(* IEC 61131-3 sources: Elmo_Master/Lasal_PRG/Elmo_EtherCAT_Test_4Axis/Class/Byte_to_Bit, 1 file *)

(* ---- Byte_to_Bit.st ---- *)
(*!
<Class
	Name               = "Byte_to_Bit"
	Revision           = "0.0"
	RealtimeTask       = "false"
	CyclicTask         = "false"
	DefCyclictime      = "1 ms"
	BackgroundTask     = "false"
	Sigmatek           = "false"
	OSInterface        = "false"
	HighPriority       = "false"
	Automatic          = "false"
	UpdateMode         = "Prescan"
	SharedCommandTable = "true"
	Objectsize         = "(300,120)">
	<Channels>
		<Server Name="bit1" Visualized="false" Initialize="false" WriteProtected="true" Retentive="false"/>
		<Server Name="bit2" Visualized="false" Initialize="false" WriteProtected="true" Retentive="false"/>
		<Server Name="bit3" Visualized="false" Initialize="false" WriteProtected="true" Retentive="false"/>
		<Server Name="bit4" Visualized="false" Initialize="false" WriteProtected="true" Retentive="false"/>
		<Server Name="bit5" Visualized="false" Initialize="false" WriteProtected="true" Retentive="false"/>
		<Server Name="bit6" Visualized="false" Initialize="false" WriteProtected="true" Retentive="false"/>
		<Server Name="bit7" Visualized="false" Initialize="false" WriteProtected="true" Retentive="false"/>
		<Server Name="bit8" Visualized="false" Initialize="false" WriteProtected="true" Retentive="false"/>
		<Server Name="ClassSvr" Visualized="false" Initialize="false" WriteProtected="true" Retentive="false"/>
		<Client Name="fromByte" Required="true" Internal="false"/>
	</Channels>
</Class>
*)
Byte_to_Bit : CLASS
  //Servers:
	ClassSvr 	: SvrChCmd_DINT;
	bit1 	: SvrCh_DINT;
	bit2 	: SvrCh_DINT;
	bit3 	: SvrCh_DINT;
	bit4 	: SvrCh_DINT;
	bit5 	: SvrCh_DINT;
	bit6 	: SvrCh_DINT;
	bit7 	: SvrCh_DINT;
	bit8 	: SvrCh_DINT;
  //Clients:
	fromByte 	: CltCh_BDINT;
  //Variables:
  //Functions:

	FUNCTION ReadByte;

	FUNCTION VIRTUAL GLOBAL bit1::Read
		VAR_OUTPUT
			output (EAX) 	: DINT;
		END_VAR;

	FUNCTION VIRTUAL GLOBAL bit2::Read
		VAR_OUTPUT
			output (EAX) 	: DINT;
		END_VAR;

	FUNCTION VIRTUAL GLOBAL bit3::Read
		VAR_OUTPUT
			output (EAX) 	: DINT;
		END_VAR;

	FUNCTION VIRTUAL GLOBAL bit4::Read
		VAR_OUTPUT
			output (EAX) 	: DINT;
		END_VAR;

	FUNCTION VIRTUAL GLOBAL bit5::Read
		VAR_OUTPUT
			output (EAX) 	: DINT;
		END_VAR;

	FUNCTION VIRTUAL GLOBAL bit6::Read
		VAR_OUTPUT
			output (EAX) 	: DINT;
		END_VAR;

	FUNCTION VIRTUAL GLOBAL bit7::Read
		VAR_OUTPUT
			output (EAX) 	: DINT;
		END_VAR;

	FUNCTION VIRTUAL GLOBAL bit8::Read
		VAR_OUTPUT
			output (EAX) 	: DINT;
		END_VAR;
  //Tables:
	FUNCTION @STD
		VAR_OUTPUT
			ret_code	: CONFSTATES;
		END_VAR;
	FUNCTION GLOBAL TAB @CT_;
END_CLASS;

FUNCTION Byte_to_Bit::ReadByte

  fromByte := fromByte.Read();

  bit1  := fromByte.1;
  bit2  := fromByte.2;
  bit3  := fromByte.3;
  bit4  := fromByte.4;
  bit5  := fromByte.5;
  bit6  := fromByte.6;
  bit7  := fromByte.7;
  bit8  := fromByte.8;

END_FUNCTION

FUNCTION VIRTUAL GLOBAL Byte_to_Bit::bit1::Read
	VAR_OUTPUT
		output (EAX) 	: DINT;
	END_VAR
  fromByte := fromByte.Read();

  bit1  := fromByte.1;
	output := bit1;

END_FUNCTION

FUNCTION VIRTUAL GLOBAL Byte_to_Bit::bit2::Read
	VAR_OUTPUT
		output (EAX) 	: DINT;
	END_VAR
  fromByte := fromByte.Read();

  bit2  := fromByte.2;
	output := bit2;

END_FUNCTION

FUNCTION VIRTUAL GLOBAL Byte_to_Bit::bit3::Read
	VAR_OUTPUT
		output (EAX) 	: DINT;
	END_VAR
  fromByte := fromByte.Read();

  bit3  := fromByte.3;
	output := bit3;

END_FUNCTION

FUNCTION VIRTUAL GLOBAL Byte_to_Bit::bit4::Read
	VAR_OUTPUT
		output (EAX) 	: DINT;
	END_VAR
  fromByte := fromByte.Read();

  bit4  := fromByte.4;
	output := bit4;

END_FUNCTION

FUNCTION VIRTUAL GLOBAL Byte_to_Bit::bit5::Read
	VAR_OUTPUT
		output (EAX) 	: DINT;
	END_VAR
  fromByte := fromByte.Read();

  bit5  := fromByte.5;
	output := bit5;

END_FUNCTION

FUNCTION VIRTUAL GLOBAL Byte_to_Bit::bit6::Read
	VAR_OUTPUT
		output (EAX) 	: DINT;
	END_VAR
  fromByte := fromByte.Read();

  bit6  := fromByte.6;
	output := bit6;

END_FUNCTION

FUNCTION VIRTUAL GLOBAL Byte_to_Bit::bit7::Read
	VAR_OUTPUT
		output (EAX) 	: DINT;
	END_VAR
  fromByte := fromByte.Read();

  bit7  := fromByte.7;
	output := bit7;

END_FUNCTION

FUNCTION VIRTUAL GLOBAL Byte_to_Bit::bit8::Read
	VAR_OUTPUT
		output (EAX) 	: DINT;
	END_VAR
  fromByte := fromByte.Read();

  bit8  := fromByte.8;
	output := bit8;

END_FUNCTION
